SUBAPPLICATION Uebung_003b_sub (* IX auf QX (generisch) *)
  (* Standard: 61499-2; Description: Copyright (c) 2023 Meisterschulen am Ostbahnhof This program and the accompanying materials are made available under the terms of the Eclipse Public License 2.0 which is available at https://www.eclipse.org/legal/epl-2.0/ SPDX-License-Identifier: EPL-2.0 *)
  (* Version 1.0, 2023-10-23, Franz Höpfinger, Meisterschulen am Ostbahnhof *)
  PACKAGE Uebungen;
  IMPORT logiBUS::io::DI::logiBUS_DI;
  IMPORT logiBUS::io::DI::logiBUS_DI_S;
  IMPORT logiBUS::io::DQ::logiBUS_DO;
  IMPORT logiBUS::io::DQ::logiBUS_DO_S;
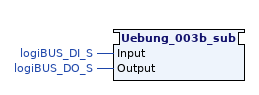
  VAR_INPUT
    Input : logiBUS::io::DI::logiBUS_DI_S := logiBUS_DI::Invalid; (* Identify the Input Input_I1..I8 *)
    Output : logiBUS::io::DQ::logiBUS_DO_S := logiBUS_DO::Invalid; (* Identify the Output Output_Q1..Q8 *)
  END_VAR
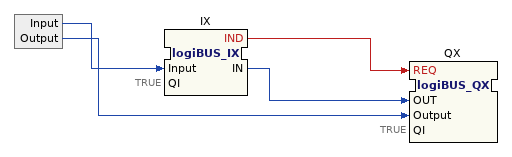
  FBS
    QX : logiBUS::io::DQ::logiBUS_QX(QI := TRUE);
    IX : logiBUS::io::DI::logiBUS_IX(QI := TRUE);
  END_FBS
  EVENT_CONNECTIONS
    IX.IND TO QX.REQ;
  END_CONNECTIONS
  DATA_CONNECTIONS
    IX.IN TO QX.OUT;
    Input TO IX.Input;
    Output TO QX.Output;
  END_CONNECTIONS
END_SUBAPPLICATION
